(* Logix 5000 project; controller WWTP_SOLIDS_CLX vendor 1 type 14 code 54 rev 17.2; software revision 17.00; part 8 of 16 *)
(* tags used below, declared in another part *)
   PCmd_Tare : BOOL;   // Program Command to Tare (reset delivered qty to 0)
   PCmd_StartFlow : BOOL;   // Program Command to Start Delivery
   PCmd_StopFlow : BOOL;   // Program Command to Stop/Pause Delivery
   PCmd_CheckTol : BOOL;   // Program Command to Check Tolerances
   PCmd_OverTolInhibit : BOOL;   // Program Command to Inhibit Out of Tolerance High Alarm
   PCmd_OverTolUninhibit : BOOL;   // Program Command to Uninhibit Out of Tolerance High Alarm
   PCmd_UnderTolInhibit : BOOL;   // Program Command to Inhibit Out of Tolerance Low Alarm
   PCmd_UnderTolUninhibit : BOOL;   // Program Command to Uninhibit Out of Tolerance Low Alarm
   PCmd_TareFaultInhibit : BOOL;   // Program Command to Inhibit Tare Fault Alarm
   PCmd_TareFaultUninhibit : BOOL;   // Program Command to Uninhibit Tare Fault Alarm
   PCmd_EqpFaultInhibit : BOOL;   // Program Command to Inhibit Equipment Fault Alarm
   PCmd_EqpFaultUninhibit : BOOL;   // Program Command to Uninhibit Equipment Fault Alarm
   OCmd_Tare : BOOL;   // Operator Command to Tare (reset delivered qty to 0)
   OCmd_StartFlow : BOOL;   // Operator command to Start Deliver
   OCmd_StopFlow : BOOL;   // Operator Command to Stop/Pause Delivery
   OCmd_CheckTol : BOOL;   // Operator Command to Check Tolerances
   OCmd_Bump : BOOL;   // Operator Command to Bump Delivery for Under Tolerance
   Rdy_Tare : BOOL;   // 1=Ready for OCmd_Tare (enables button)
   Rdy_StartFlow : BOOL;   // 1=Ready for OCmd_StartFlow (enables button)
   Rdy_StopFlow : BOOL;   // 1=Ready for OCmd_StopFlow (enables button)
   Rdy_CheckTol : BOOL;   // 1-Ready for OCmd_CheckTol (enables button)
   Rdy_Bump : BOOL;   // 1=Ready for OCmd_Bump (enables button)
   Wrk_ValidONS1 : BOOL;   // Weight PV goes from Infinite or Not a Number to VALID
   Wrk_ValidONS2 : BOOL;   // Rate goes from Infinite or Not a Number to VALID
(* P_DoseWS, continued *)

ROUTINE Prescan   (* ladder *)
// Clear Ownership, clear "lurking" Commands, all Readies
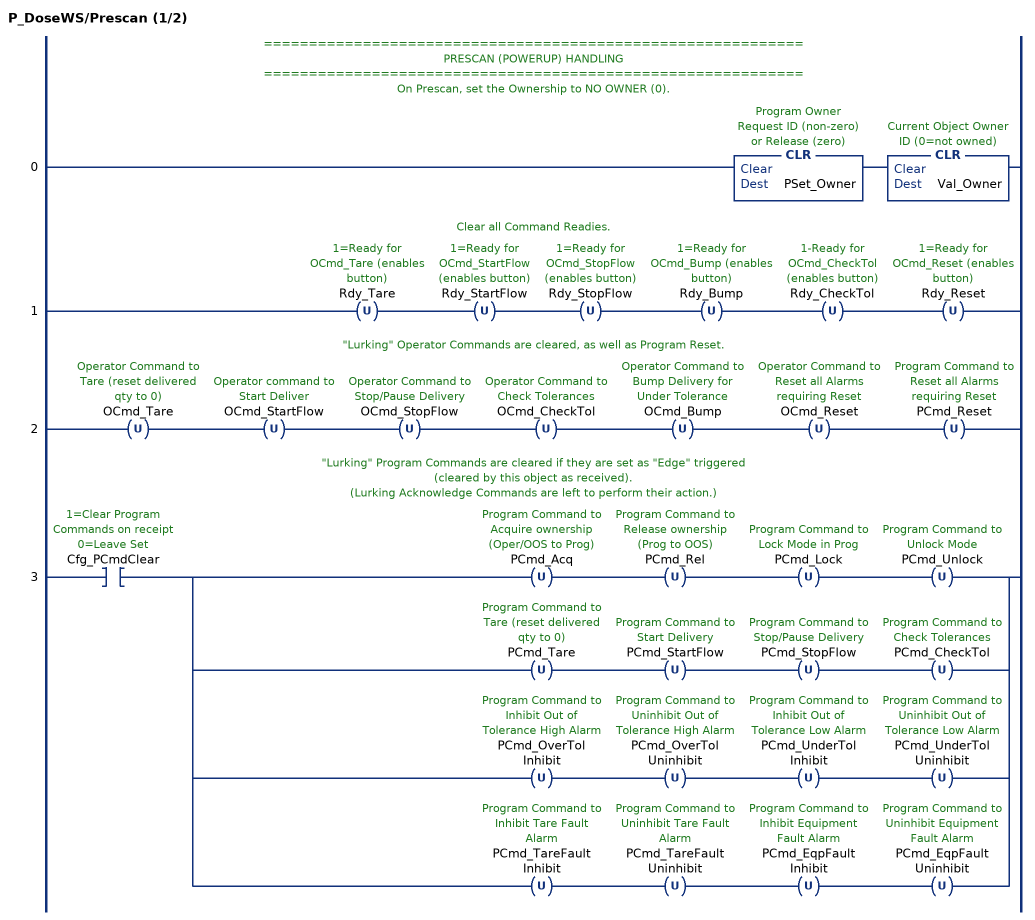
   // ============================================================
   // PRESCAN (POWERUP) HANDLING
   // ============================================================
   // On Prescan, set the Ownership to NO OWNER (0).
   0: CLR(PSet_Owner)CLR(Val_Owner);
   // Clear all Command Readies.
   1: OTU(Rdy_Tare)OTU(Rdy_StartFlow)OTU(Rdy_StopFlow)OTU(Rdy_Bump)OTU(Rdy_CheckTol)OTU(Rdy_Reset);
   // "Lurking" Operator Commands are cleared, as well as Program Reset.
   2: OTU(OCmd_Tare)OTU(OCmd_StartFlow)OTU(OCmd_StopFlow)OTU(OCmd_CheckTol)OTU(OCmd_Bump)OTU(OCmd_Reset)OTU(PCmd_Reset);
   // "Lurking" Program Commands are cleared if they are set as "Edge" triggered
   // (cleared by this object as received).
   // (Lurking Acknowledge Commands are left to perform their action.)
   3: XIC(Cfg_PCmdClear)[OTU(PCmd_Acq) OTU(PCmd_Rel) OTU(PCmd_Lock) OTU(PCmd_Unlock) ,OTU(PCmd_Tare) OTU(PCmd_StartFlow) OTU(PCmd_StopFlow) OTU(PCmd_CheckTol) ,OTU(PCmd_OverTolInhibit) OTU(PCmd_OverTolUninhibit) OTU(PCmd_UnderTolInhibit) OTU(PCmd_UnderTolUninhibit) ,OTU(PCmd_TareFaultInhibit) OTU(PCmd_TareFaultUninhibit) OTU(PCmd_EqpFaultInhibit) OTU(PCmd_EqpFaultUninhibit) ];
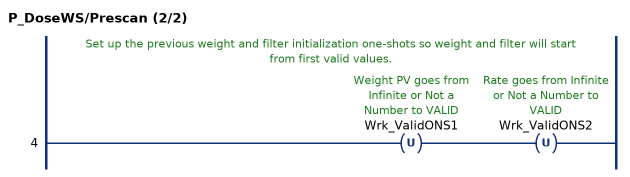
   // Set up the previous weight and filter initialization one-shots so weight and filter will start from first valid values.
   4: OTU(Wrk_ValidONS1)OTU(Wrk_ValidONS2);
END_ROUTINE
END_ADD_ON_INSTRUCTION

ADD_ON_INSTRUCTION P_Intlk   (* revision 0.10, ExecuteEnableInFalse *)
// Interlocks
// Revision note:
// Aligned name, description and local STRING values, sizes, across instructions.
// Help:
// This Instruction monitors up to 16 Interlock conditions.  It provides these features:
// *  Interlocks may be configured as Latched.
//     Latched Interlocks require a Reset Command to clear.
// *  Interlocks may be configured as Bypassable; Non-Bypassable
//     Interlocks are reported separately so the destination object can
//     decide whether to bypass (ignore) bypassable interlocks, such
//     as in Maintenance Mode.
// *  First-Out reporting indicates the first condition that caused the
//     running equipment to be tripped.  A separate First-Out is provided
//     for Non-Bypassable Interlocks.
VAR_INPUT
   Inp_Intlk00 : BOOL; {visible}   // Interlock Cond. 00 (1=Stop, 0=OK)
   Inp_Intlk01 : BOOL; {visible}   // Interlock Cond. 01 (1=Stop, 0=OK)
   Inp_Intlk02 : BOOL; {visible}   // Interlock Cond. 02 (1=Stop, 0=OK)
   Inp_Intlk03 : BOOL; {visible}   // Interlock Cond. 03 (1=Stop, 0=OK)
   Inp_Intlk04 : BOOL; {visible}   // Interlock Cond. 04 (1=Stop, 0=OK)
   Inp_Intlk05 : BOOL; {visible}   // Interlock Cond. 05 (1=Stop, 0=OK)
   Inp_Intlk06 : BOOL; {visible}   // Interlock Cond. 06 (1=Stop, 0=OK)
   Inp_Intlk07 : BOOL; {visible}   // Interlock Cond. 07 (1=Stop, 0=OK)
   Inp_Intlk08 : BOOL;   // Interlock Cond. 08 (1=Stop, 0=OK)
   Inp_Intlk09 : BOOL;   // Interlock Cond. 09 (1=Stop, 0=OK)
   Inp_Intlk10 : BOOL;   // Interlock Cond. 10 (1=Stop, 0=OK)
   Inp_Intlk11 : BOOL;   // Interlock Cond. 11 (1=Stop, 0=OK)
   Inp_Intlk12 : BOOL;   // Interlock Cond. 12 (1=Stop, 0=OK)
   Inp_Intlk13 : BOOL;   // Interlock Cond. 13 (1=Stop, 0=OK)
   Inp_Intlk14 : BOOL;   // Interlock Cond. 14 (1=Stop, 0=OK)
   Inp_Intlk15 : BOOL;   // Interlock Cond. 15 (1=Stop, 0=OK)
   Inp_Reset : BOOL; {visible}   // 1=Reset Latched Interlocks and First-Out
   Cfg_Latched : INT;   // Set bits indicate which conditions are latched (sealed in)
   Cfg_Bypassable : INT;   // Set bits indicate which conditions can be bypassed
   Cfg_PCmdClear : BOOL := 1;   // 1=Clear Program Commands on receipt 0=Leave Set
   PCmd_Reset : BOOL;   // Program Command to Reset Latched Interlocks
   OCmd_Reset : BOOL;   // Operator Command to Reset Latched Interlocks
END_VAR
VAR_OUTPUT
   Sts_IntlkOK : BOOL := 1; {visible}   // Overall Interlock Status (1=OK to run, 0=Stop)
   Sts_NBIntlkOK : BOOL := 1; {visible}   // Non-Bypassable Interlock Status (1=All NB Interlocks OK to run)
   Sts_Intlk : INT; {visible}   // Individual Interlock Status (1=Stop, 0=OK)
   Sts_FirstOut : INT; {visible}   // Interlock First Out Status (bit 1 is First Not-OK condition)
   Sts_NBFirstOut : INT; {visible}   // Non-bypassable Interlock First-Out Status (bit=1 is First NB Not-OK condition)
   Rdy_Reset : BOOL;   // 1=Ready to receive OCmd_Reset (reset required)
END_VAR
VAR
   Cfg_CondTxt : STRING_20[16] := ([0] := 'Interlock 0');   // Short HMI description of Interlock Conditions
   Wrk_Inp : INT;   // Collection copy of Inp_IntlkXXs
   Wrk_NB : INT;   // Working register for Non-Bypassable Interlock ogic
   Wrk_Intlk : INT;   // Working register for Interlock logic
   Wrk_FirstOut : INT;   // Working register for First Out logic
   Wrk_Sts : INT;   // Working register for generating Interlock status
   Wrk_NBFirstOut : INT;   // Working register for Non-Bypassable First Out logic
   Wrk_PrevSts : INT;   // Interlock Status previous scan
   Wrk_PrevNB : INT;   // Non-Bypassable Status previous scan
END_VAR

ROUTINE EnableInFalse   (* ladder *)
// Set summary "OK" Status bits to FALSE (0)
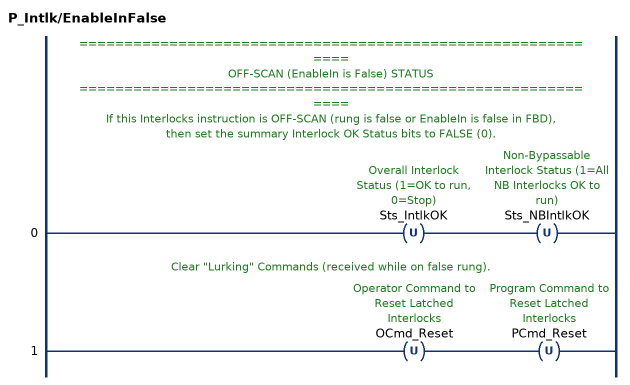
   // ============================================================
   // OFF-SCAN (EnableIn is False) STATUS
   // ============================================================
   // If this Interlocks instruction is OFF-SCAN (rung is false or EnableIn is false in FBD),
   // then set the summary Interlock OK Status bits to FALSE (0).
   0: OTU(Sts_IntlkOK)OTU(Sts_NBIntlkOK);
   // Clear "Lurking" Commands (received while on false rung).
   1: OTU(OCmd_Reset)OTU(PCmd_Reset);
END_ROUTINE

ROUTINE Logic   (* ladder *)
// Check Interlock Conditions
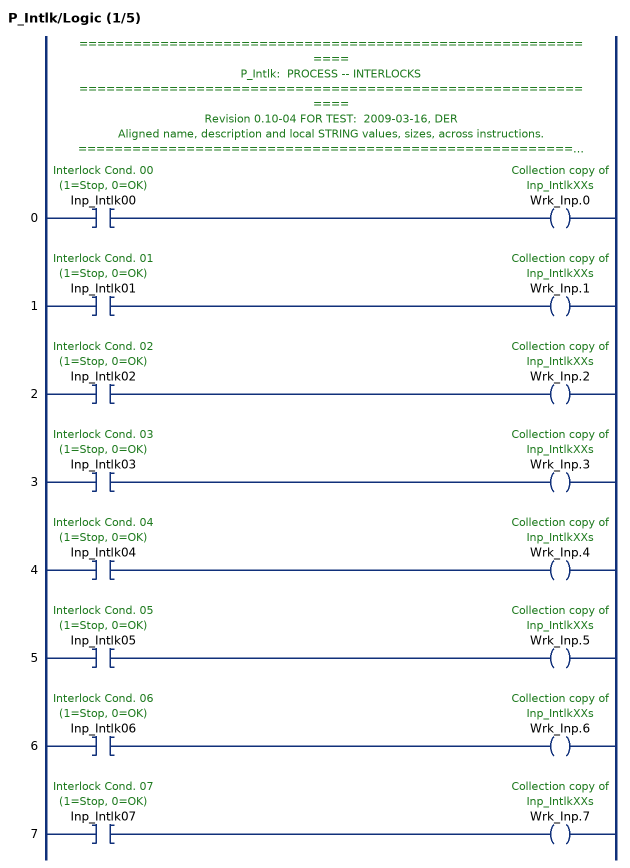
   // ============================================================
   // P_Intlk:  PROCESS -- INTERLOCKS
   // ============================================================
   // Revision 0.10-04 FOR TEST:  2009-03-16, DER
   // Aligned name, description and local STRING values, sizes, across instructions.
   // ============================================================
   // This Instruction monitors up to 16 Interlock conditions.  It provides these features:
   // *  Interlocks may be configured as Latched.  Latched Interlocks
   // require a Reset Command to clear.
   // *  Interlocks may be configured as Bypassable.  Bypassable Interlocks are reported
   // separately; the destination object can use this information to bypass these
   // Interlocks in Maintenance Mode or upon command.
   // *  First-Out reporting indicates the first condition that caused the running equipment
   // to be tripped.  Separate First-Out for Non-Bypassable Interlocks.
   // ============================================================
   // POWERUP / INVALID STATE HANDLING
   // ============================================================
   // Interlock, bypass and lock states are maintained through a power cycle or
   // run/prog/run cycle. No special powerup code is required for this object.
   // ============================================================
   // INPUT GATHERING
   // ============================================================
   // This object uses word-wise logic.  The first 16 rungs collect the individual
   // Interlock Inputs together into a 16-bit integer word for word-wise processing.
   0: XIC(Inp_Intlk00)OTE(Wrk_Inp.0);
   1: XIC(Inp_Intlk01)OTE(Wrk_Inp.1);
   2: XIC(Inp_Intlk02)OTE(Wrk_Inp.2);
   3: XIC(Inp_Intlk03)OTE(Wrk_Inp.3);
   4: XIC(Inp_Intlk04)OTE(Wrk_Inp.4);
   5: XIC(Inp_Intlk05)OTE(Wrk_Inp.5);
   6: XIC(Inp_Intlk06)OTE(Wrk_Inp.6);
   7: XIC(Inp_Intlk07)OTE(Wrk_Inp.7);
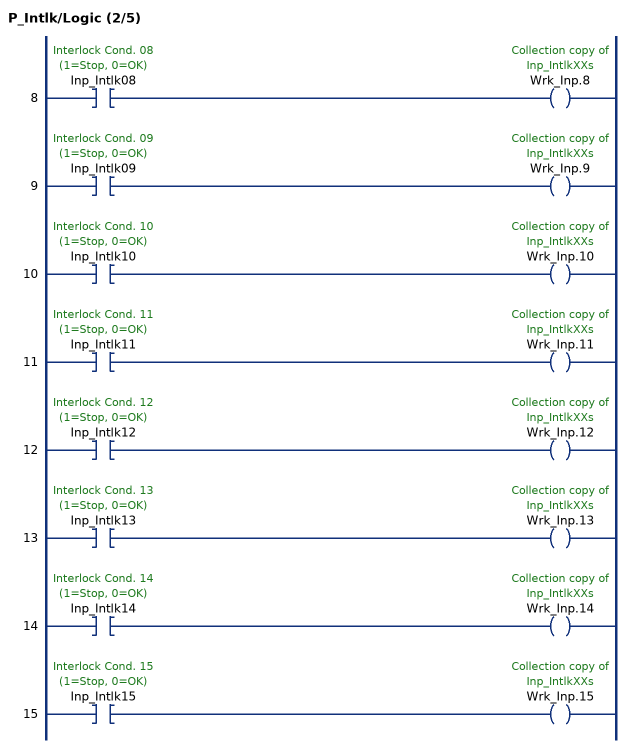
   8: XIC(Inp_Intlk08)OTE(Wrk_Inp.8);
   9: XIC(Inp_Intlk09)OTE(Wrk_Inp.9);
   10: XIC(Inp_Intlk10)OTE(Wrk_Inp.10);
   11: XIC(Inp_Intlk11)OTE(Wrk_Inp.11);
   12: XIC(Inp_Intlk12)OTE(Wrk_Inp.12);
   13: XIC(Inp_Intlk13)OTE(Wrk_Inp.13);
   14: XIC(Inp_Intlk14)OTE(Wrk_Inp.14);
   15: XIC(Inp_Intlk15)OTE(Wrk_Inp.15);
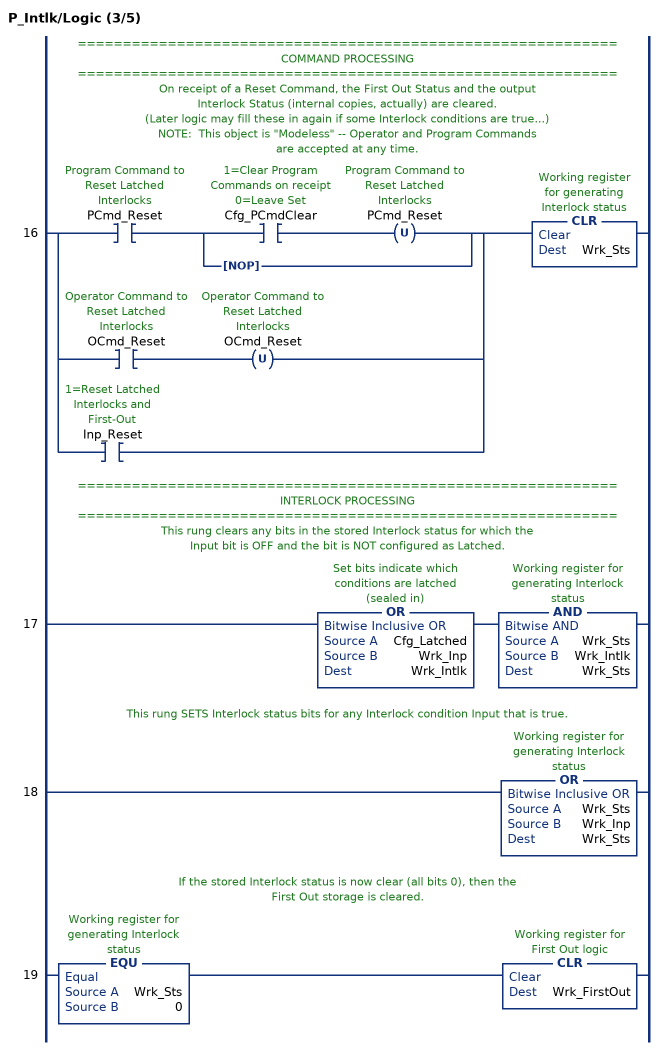
   // ============================================================
   // COMMAND PROCESSING
   // ============================================================
   // On receipt of a Reset Command, the First Out Status and the output
   // Interlock Status (internal copies, actually) are cleared.
   // (Later logic may fill these in again if some Interlock conditions are true...)
   // NOTE:  This object is "Modeless" -- Operator and Program Commands
   // are accepted at any time.
   16: [XIC(PCmd_Reset) [XIC(Cfg_PCmdClear) OTU(PCmd_Reset) ,NOP() ] ,XIC(OCmd_Reset) OTU(OCmd_Reset) ,XIC(Inp_Reset) ]CLR(Wrk_Sts);
   // ============================================================
   // INTERLOCK PROCESSING
   // ============================================================
   // This rung clears any bits in the stored Interlock status for which the
   // Input bit is OFF and the bit is NOT configured as Latched.
   17: OR(Cfg_Latched,Wrk_Inp,Wrk_Intlk)AND(Wrk_Sts,Wrk_Intlk,Wrk_Sts);
   // This rung SETS Interlock status bits for any Interlock condition Input that is true.
   18: OR(Wrk_Sts,Wrk_Inp,Wrk_Sts);
   // If the stored Interlock status is now clear (all bits 0), then the
   // First Out storage is cleared.
   19: EQU(Wrk_Sts,0)CLR(Wrk_FirstOut);
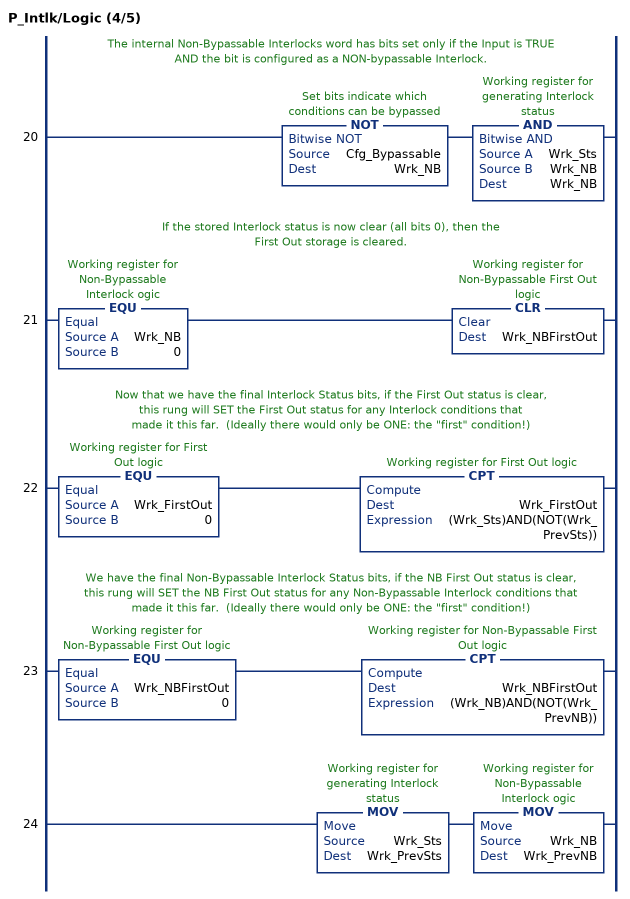
   // The internal Non-Bypassable Interlocks word has bits set only if the Input is TRUE
   // AND the bit is configured as a NON-bypassable Interlock.
   20: NOT(Cfg_Bypassable,Wrk_NB)AND(Wrk_Sts,Wrk_NB,Wrk_NB);
   // If the stored Interlock status is now clear (all bits 0), then the
   // First Out storage is cleared.
   21: EQU(Wrk_NB,0)CLR(Wrk_NBFirstOut);
   // Now that we have the final Interlock Status bits, if the First Out status is clear,
   // this rung will SET the First Out status for any Interlock conditions that
   // made it this far.  (Ideally there would only be ONE: the "first" condition!)
   22: EQU(Wrk_FirstOut,0)CPT(Wrk_FirstOut,(Wrk_Sts)AND(NOT(Wrk_PrevSts)));
   // We have the final Non-Bypassable Interlock Status bits, if the NB First Out status is clear,
   // this rung will SET the NB First Out status for any Non-Bypassable Interlock conditions that
   // made it this far.  (Ideally there would only be ONE: the "first" condition!)
   23: EQU(Wrk_NBFirstOut,0)CPT(Wrk_NBFirstOut,(Wrk_NB)AND(NOT(Wrk_PrevNB)));
   24: MOV(Wrk_Sts,Wrk_PrevSts)MOV(Wrk_NB,Wrk_PrevNB);
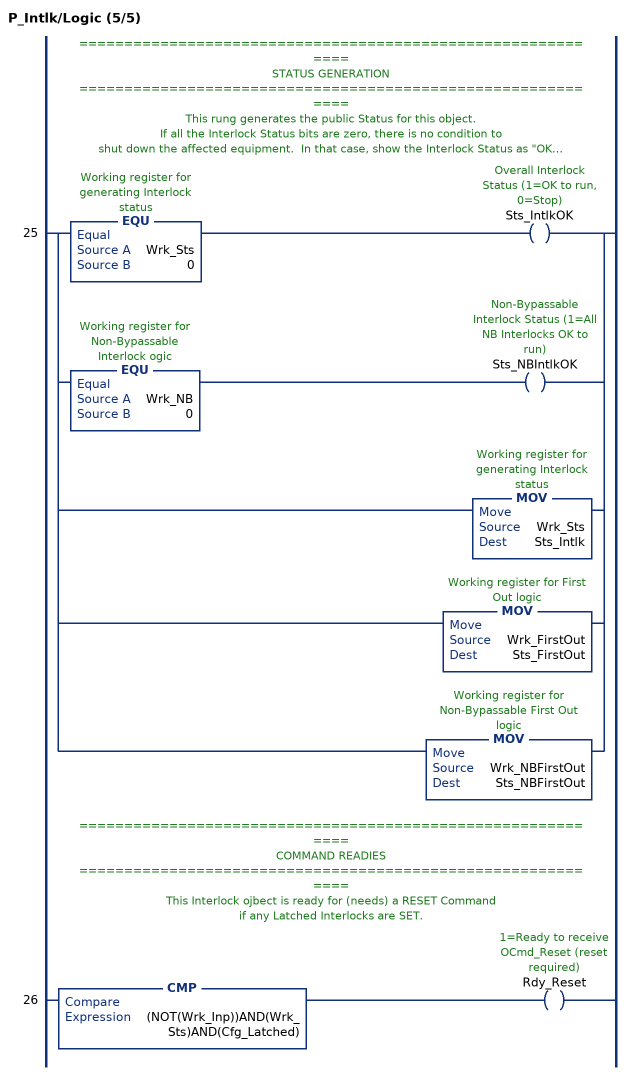
   // ============================================================
   // STATUS GENERATION
   // ============================================================
   // This rung generates the public Status for this object.
   // If all the Interlock Status bits are zero, there is no condition to
   // shut down the affected equipment.  In that case, show the Interlock Status as "OK"
   // Similar logic applies for the Non-Bypassable Interlocks OK Status.
   // Also show the individual Interlock Status bits and the First Out Status bits.
   // NOTE:  Working registers are used to prevent outside writes to the Sts_xxx
   // parameters from affecting the state of this object!
   25: [[EQU(Wrk_Sts,0) OTE(Sts_IntlkOK) ,EQU(Wrk_NB,0) OTE(Sts_NBIntlkOK) ] ,MOV(Wrk_Sts,Sts_Intlk) ,MOV(Wrk_FirstOut,Sts_FirstOut) ,MOV(Wrk_NBFirstOut,Sts_NBFirstOut) ];
   // ============================================================
   // COMMAND READIES
   // ============================================================
   // This Interlock ojbect is ready for (needs) a RESET Command
   // if any Latched Interlocks are SET.
   26: CMP((NOT(Wrk_Inp))AND(Wrk_Sts)AND(Cfg_Latched))OTE(Rdy_Reset);
END_ROUTINE

ROUTINE Prescan   (* ladder *)
// Clear "lurking" Commands
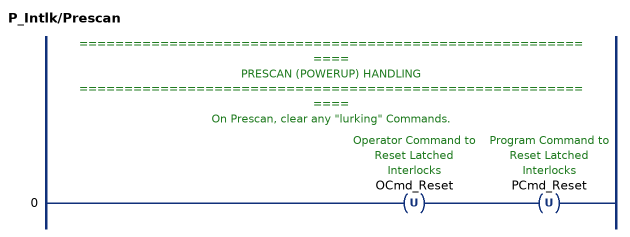
   // ============================================================
   // PRESCAN (POWERUP) HANDLING
   // ============================================================
   // On Prescan, clear any "lurking" Commands.
   0: OTU(OCmd_Reset)OTU(PCmd_Reset);
END_ROUTINE
END_ADD_ON_INSTRUCTION

ADD_ON_INSTRUCTION P_Mode   (* revision 0.20, ExecutePrescan, ExecuteEnableInFalse *)
// Mode
// Revision note:
// Aligned name, description and local STRING values, sizes, across instructions.
// Help:
// This instruction provides selection of Mode for a Device-level
//  object (motor, valve, drive, loop, etc.).  Possible Modes are:
//    Hand (typically tracks hardwired logic)
//    Maintenance (not available for operation)
//    Override (typically process or soft safety interlock logic)
//    Operator (settings and commands from HMI)
//    Program (settings and commands from other objects)
// Hand and Override are selected via Input parameters (pins).
// Program and Maintenance are acquired and released via Commands.
// Program or Operator owner can Lock ownership; when locked, Hand and
// Maintenance override the Lock.  Override can be configured as to
// whether or not it supersedes Locked Program or Operator ownership.
// Program Commands can be configured as one-shot (OTL) inputs (default),
// or Level-based inputs.  One-shot Program Commands are cleared by the
// Mode object; When Level-based, the Program Acquire (PCmd_Acq)
// Command is left set; when the Program clears this Command, Program Mode is
// released; and when the Program Lock (PCmd_Lock) command is cleared,
// Program Mode is unlocked.
// Program and Operator commands work "behind the scenes" while in Hand,
// Ovrd or Maint; so the Program can release the object while in Hand, and
// upon exiting Hand, the Mode will revert to Operator, for example.  Extra Status
// bits indicate the results of these "behind the scenes" activities.
VAR_INPUT
   Inp_Hand : BOOL; {visible}   // 1=Select Hand (typ. hardwired) Mode
   Inp_Ovrd : BOOL; {visible}   // 1=Select Override (typ. Process/Safety Interlock) Mode
   Cfg_PCmdClear : BOOL := 1;   // 1=Clear Program Command on receipt; 0=Use Level-based (maintained) PCmds
   Cfg_OvrdOverLock : BOOL := 1;   // 1=Override supersedes Prog/Oper Lock, 0=don't override Lock
   PCmd_Acq : BOOL;   // Program Command to Acquire Ownership (Oper to Prog)
   PCmd_Rel : BOOL;   // Program Command to Release Ownership (Prog to Oper)
   PCmd_Lock : BOOL;   // Program Command to Lock Mode in Prog
   PCmd_Unlock : BOOL;   // Program Command to Unlock Mode
   MCmd_Acq : BOOL;   // Maintenance Command to Acquire Ownership (Oper/Prog/Ovrd to Maint)
   MCmd_Rel : BOOL;   // Maintenance Command to Release Ownership (Maint to Oper/Prog/Ovrd)
   OCmd_AcqLock : BOOL;   // Operator Command to Acquire and Lock Mode in Oper
   OCmd_Unlock : BOOL;   // Operator Command to Unlock Operator Mode
END_VAR
VAR_OUTPUT
   Sts_Hand : BOOL; {visible}   // 1=Mode is Hand (supersedes Maint, Ovrd, Prog, Oper)
   Sts_Maint : BOOL; {visible}   // 1=Mode is Maintenance (supersedes Ovrd, Prog, Oper)
   Sts_Ovrd : BOOL; {visible}   // 1=Mode is Override (supersedes Prog, Oper)
   Sts_Prog : BOOL; {visible}   // 1=Mode is Program
   Sts_Oper : BOOL := 1; {visible}   // 1=Mode is Operator
   Sts_ProgOperLock : BOOL; {visible}   // 1=Program or Operator has requested Mode Lock
   Sts_ProgOperSel : BOOL;   // Prog/Oper selection 1=Program, 0=Operator
   Rdy_Acq : BOOL;   // 1=Ready for MCmd_Acq
   Rdy_Rel : BOOL;   // 1=Ready for MCmd_Rel
   Rdy_AcqLock : BOOL;   // 1=Ready for OCmd_AcqLock
   Rdy_Unlock : BOOL;   // 1=Ready for OCmd_Unlock
END_VAR
VAR
   Wrk_Locked : BOOL;   // 1=Program/Operator Mode selection is Locked
   Wrk_Prog : BOOL;   // Internal Program (1) / Operator (0) Mode selection
   Wrk_Maint : BOOL;   // Internal Maintenance Mode
END_VAR

ROUTINE EnableInFalse   (* ladder *)
// Processes received Commands, but shows NO owner
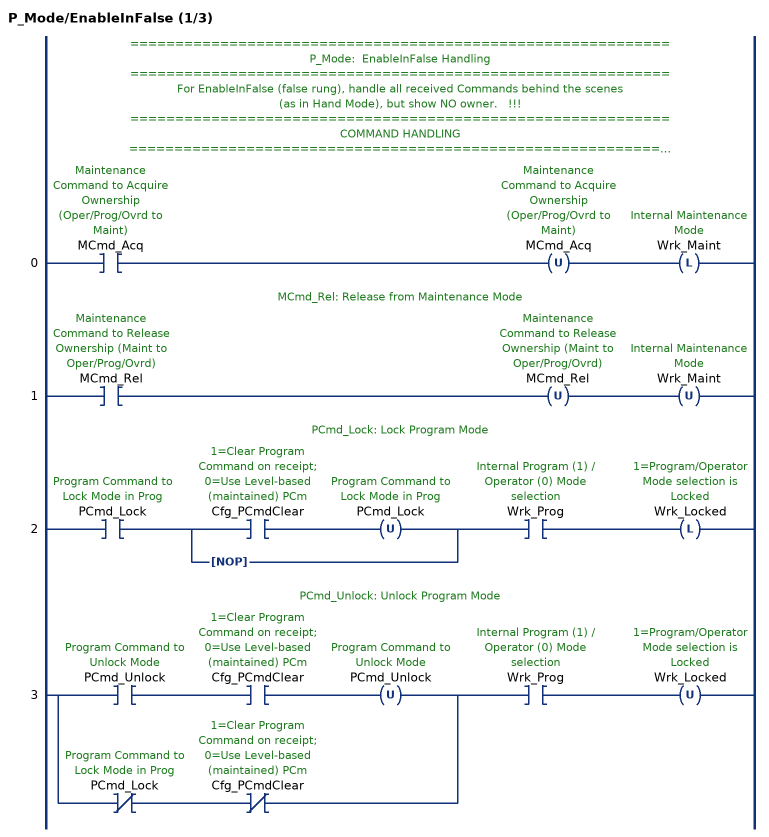
   // ============================================================
   // P_Mode:  EnableInFalse Handling
   // ============================================================
   // For EnableInFalse (false rung), handle all received Commands behind the scenes
   // (as in Hand Mode), but show NO owner.   !!!
   // ============================================================
   // COMMAND HANDLING
   // ============================================================
   // NOTE:  These rungs MUST be in the order given to meet the following
   // multiple-actions-at-the-same-time scenarios:
   // * Maintenance Release beats Maintenance Acquire
   // * Program Release beats Program Acquire
   // * Program Unlock beats Program Lock
   // * Operator Unlock beats Operator Acquire and Lock (results in Oper Unlocked)
   // * Operator Acquire/Lock must come after Program Unlock
   // * Program Acquire must come after Operator Unlock
   // MCmd_Acq: Acquire for Maintenance Mode
   0: XIC(MCmd_Acq)OTU(MCmd_Acq)OTL(Wrk_Maint);
   // MCmd_Rel: Release from Maintenance Mode
   1: XIC(MCmd_Rel)OTU(MCmd_Rel)OTU(Wrk_Maint);
   // PCmd_Lock: Lock Program Mode
   2: XIC(PCmd_Lock)[XIC(Cfg_PCmdClear) OTU(PCmd_Lock) ,NOP() ]XIC(Wrk_Prog)OTL(Wrk_Locked);
   // PCmd_Unlock: Unlock Program Mode
   3: [XIC(PCmd_Unlock) XIC(Cfg_PCmdClear) OTU(PCmd_Unlock) ,XIO(PCmd_Lock) XIO(Cfg_PCmdClear) ]XIC(Wrk_Prog)OTU(Wrk_Locked);
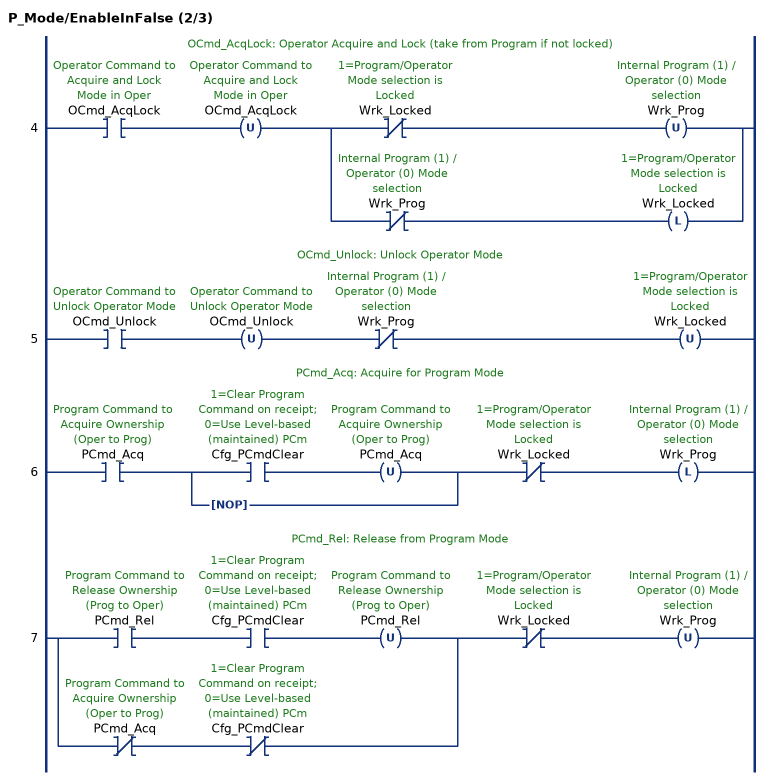
   // OCmd_AcqLock: Operator Acquire and Lock (take from Program if not locked)
   4: XIC(OCmd_AcqLock)OTU(OCmd_AcqLock)[XIO(Wrk_Locked) OTU(Wrk_Prog) ,XIO(Wrk_Prog) OTL(Wrk_Locked) ];
   // OCmd_Unlock: Unlock Operator Mode
   5: XIC(OCmd_Unlock)OTU(OCmd_Unlock)XIO(Wrk_Prog)OTU(Wrk_Locked);
   // PCmd_Acq: Acquire for Program Mode
   6: XIC(PCmd_Acq)[XIC(Cfg_PCmdClear) OTU(PCmd_Acq) ,NOP() ]XIO(Wrk_Locked)OTL(Wrk_Prog);
   // PCmd_Rel: Release from Program Mode
   7: [XIC(PCmd_Rel) XIC(Cfg_PCmdClear) OTU(PCmd_Rel) ,XIO(PCmd_Acq) XIO(Cfg_PCmdClear) ]XIO(Wrk_Locked)OTU(Wrk_Prog);
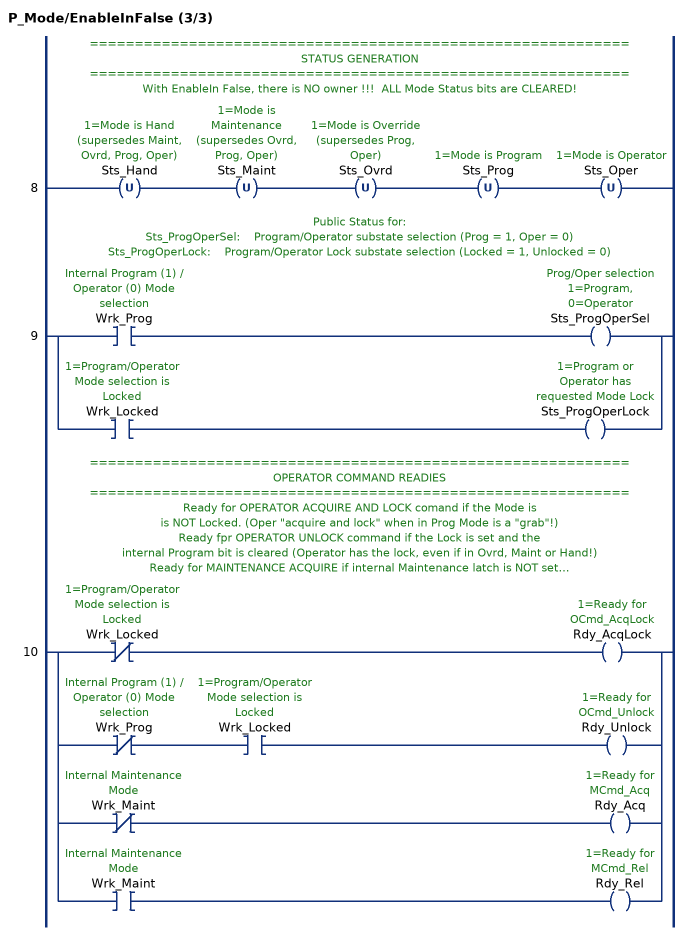
   // ============================================================
   // STATUS GENERATION
   // ============================================================
   // With EnableIn False, there is NO owner !!!  ALL Mode Status bits are CLEARED!
   8: OTU(Sts_Hand)OTU(Sts_Maint)OTU(Sts_Ovrd)OTU(Sts_Prog)OTU(Sts_Oper);
   // Public Status for:
   // Sts_ProgOperSel:    Program/Operator substate selection (Prog = 1, Oper = 0)
   // Sts_ProgOperLock:    Program/Operator Lock substate selection (Locked = 1, Unlocked = 0)
   9: [XIC(Wrk_Prog) OTE(Sts_ProgOperSel) ,XIC(Wrk_Locked) OTE(Sts_ProgOperLock) ];
   // ============================================================
   // OPERATOR COMMAND READIES
   // ============================================================
   // Ready for OPERATOR ACQUIRE AND LOCK comand if the Mode is
   //  is NOT Locked. (Oper "acquire and lock" when in Prog Mode is a "grab"!)
   // Ready fpr OPERATOR UNLOCK command if the Lock is set and the
   // internal Program bit is cleared (Operator has the lock, even if in Ovrd, Maint or Hand!)
   // Ready for MAINTENANCE ACQUIRE if internal Maintenance latch is NOT set.
   // Ready for MAINTENANCE RELEASE if internal Maintenance latch IS set.
   10: [XIO(Wrk_Locked) OTE(Rdy_AcqLock) ,XIO(Wrk_Prog) XIC(Wrk_Locked) OTE(Rdy_Unlock) ,XIO(Wrk_Maint) OTE(Rdy_Acq) ,XIC(Wrk_Maint) OTE(Rdy_Rel) ];
END_ROUTINE

ROUTINE Logic   (* ladder *)
// Selects Modes (Hand, Maint, Ovrd, Oper, Prog) based on Inputs and Commands
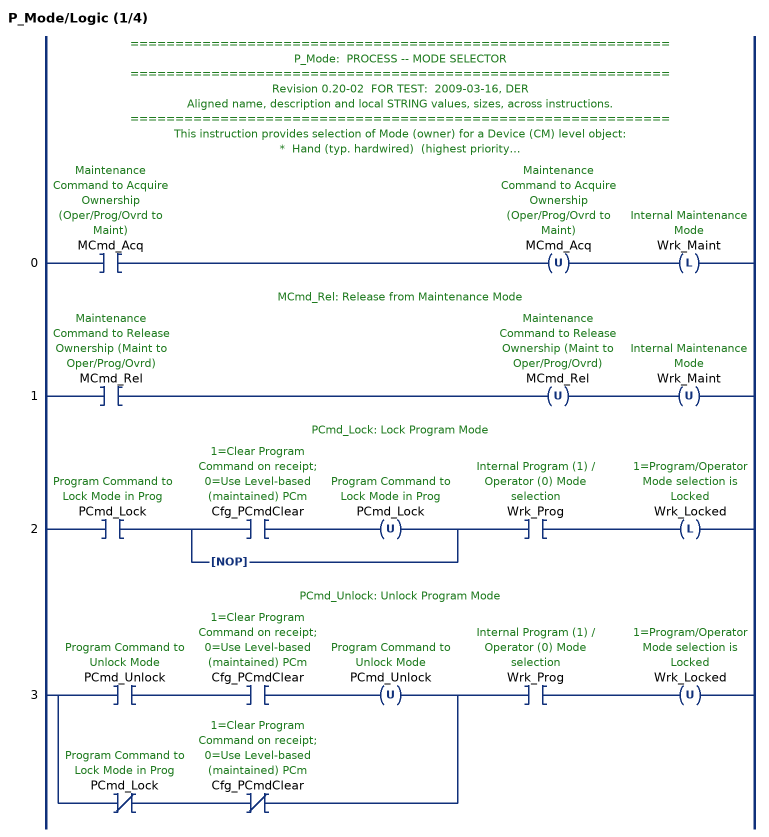
   // ============================================================
   // P_Mode:  PROCESS -- MODE SELECTOR
   // ============================================================
   // Revision 0.20-02  FOR TEST:  2009-03-16, DER
   // Aligned name, description and local STRING values, sizes, across instructions.
   // ============================================================
   // This instruction provides selection of Mode (owner) for a Device (CM) level object:
   // *  Hand (typ. hardwired)  (highest priority)
   // *  Maint (taken out of service for maintenance)
   // *  Ovrd (typ. process or soft safety interlock)
   // *  Prog  (automated control)
   // *  Oper (manual control)  (lowest priority owner)
   // ============================================================
   // COMMAND HANDLING
   // ============================================================
   // NOTE:  These rungs MUST be in the order given to meet the following
   // multiple-actions-at-the-same-time scenarios:
   // * Maintenance Release beats Maintenance Acquire
   // * Program Release beats Program Acquire
   // * Program Unlock beats Program Lock
   // * Operator Unlock beats Operator Acquire and Lock (results in Oper Unlocked)
   // * Operator Acquire/Lock must come after Program Unlock
   // * Program Acquire must come after Operator Unlock
   // MCmd_Acq: Acquire for Maintenance Mode
   0: XIC(MCmd_Acq)OTU(MCmd_Acq)OTL(Wrk_Maint);
   // MCmd_Rel: Release from Maintenance Mode
   1: XIC(MCmd_Rel)OTU(MCmd_Rel)OTU(Wrk_Maint);
   // PCmd_Lock: Lock Program Mode
   2: XIC(PCmd_Lock)[XIC(Cfg_PCmdClear) OTU(PCmd_Lock) ,NOP() ]XIC(Wrk_Prog)OTL(Wrk_Locked);
   // PCmd_Unlock: Unlock Program Mode
   3: [XIC(PCmd_Unlock) XIC(Cfg_PCmdClear) OTU(PCmd_Unlock) ,XIO(PCmd_Lock) XIO(Cfg_PCmdClear) ]XIC(Wrk_Prog)OTU(Wrk_Locked);
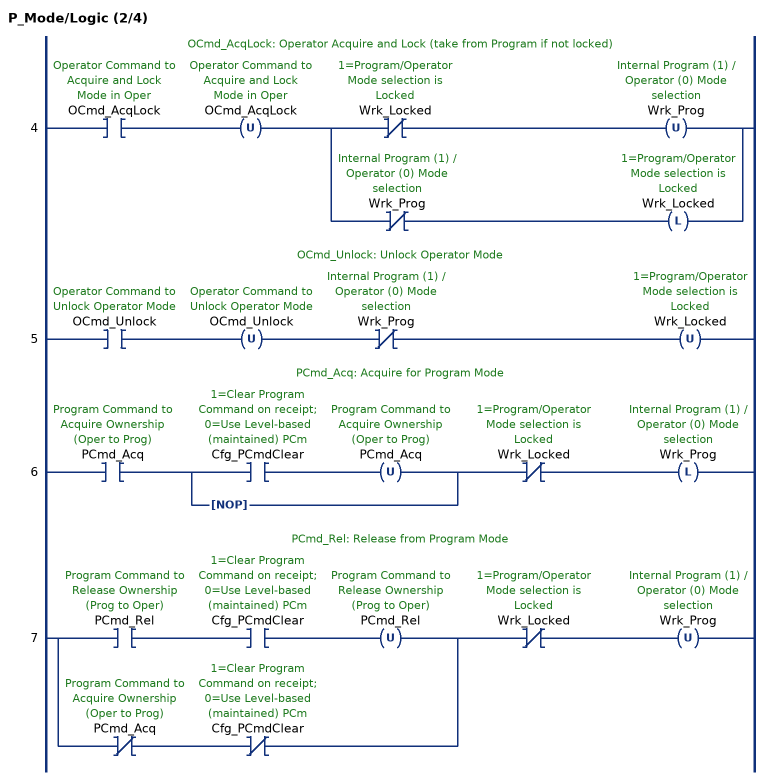
   // OCmd_AcqLock: Operator Acquire and Lock (take from Program if not locked)
   4: XIC(OCmd_AcqLock)OTU(OCmd_AcqLock)[XIO(Wrk_Locked) OTU(Wrk_Prog) ,XIO(Wrk_Prog) OTL(Wrk_Locked) ];
   // OCmd_Unlock: Unlock Operator Mode
   5: XIC(OCmd_Unlock)OTU(OCmd_Unlock)XIO(Wrk_Prog)OTU(Wrk_Locked);
   // PCmd_Acq: Acquire for Program Mode
   6: XIC(PCmd_Acq)[XIC(Cfg_PCmdClear) OTU(PCmd_Acq) ,NOP() ]XIO(Wrk_Locked)OTL(Wrk_Prog);
   // PCmd_Rel: Release from Program Mode
   7: [XIC(PCmd_Rel) XIC(Cfg_PCmdClear) OTU(PCmd_Rel) ,XIO(PCmd_Acq) XIO(Cfg_PCmdClear) ]XIO(Wrk_Locked)OTU(Wrk_Prog);
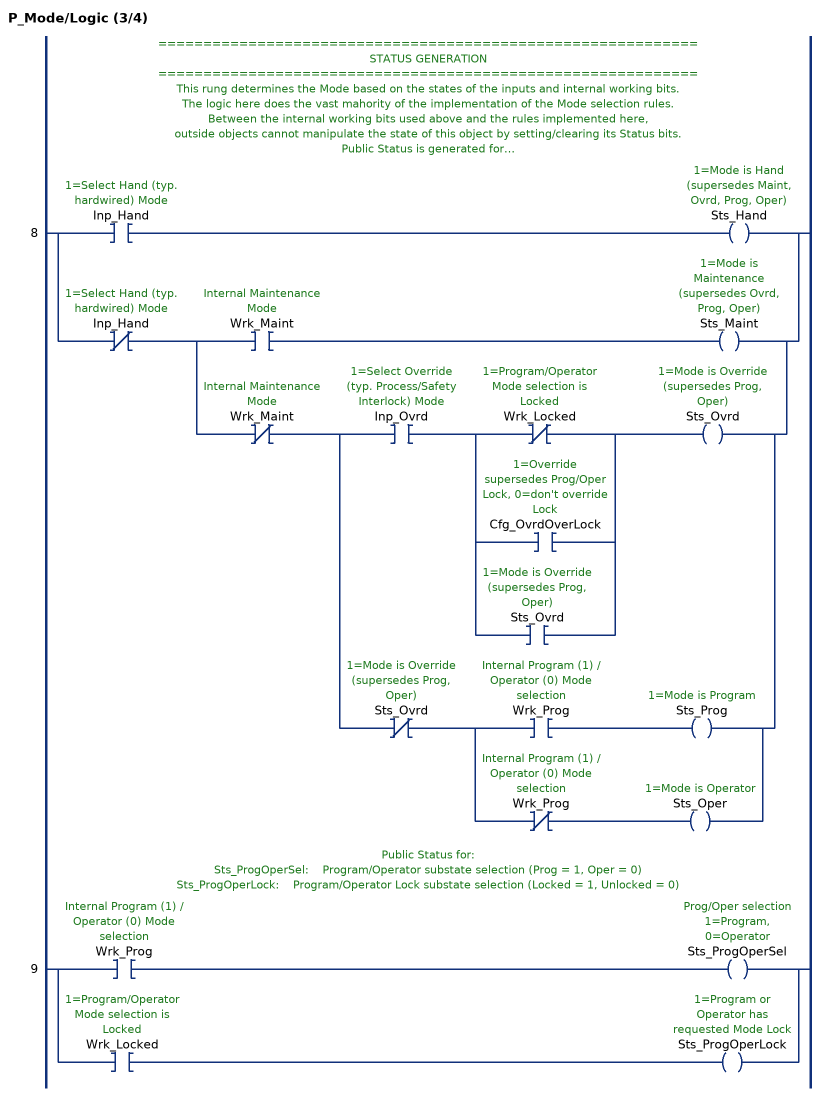
   // ============================================================
   // STATUS GENERATION
   // ============================================================
   // This rung determines the Mode based on the states of the inputs and internal working bits.
   // The logic here does the vast mahority of the implementation of the Mode selection rules.
   // Between the internal working bits used above and the rules implemented here,
   // outside objects cannot manipulate the state of this object by setting/clearing its Status bits.
   // Public Status is generated for:
   // *  Hand Mode
   // *  Maintenance Mode
   // *  Override Mode
   // *  Program Mode
   // *  Operator Mode
   8: [XIC(Inp_Hand) OTE(Sts_Hand) ,XIO(Inp_Hand) [XIC(Wrk_Maint) OTE(Sts_Maint) ,XIO(Wrk_Maint) [XIC(Inp_Ovrd) [XIO(Wrk_Locked) ,XIC(Cfg_OvrdOverLock) ,XIC(Sts_Ovrd) ] OTE(Sts_Ovrd) ,XIO(Sts_Ovrd) [XIC(Wrk_Prog) OTE(Sts_Prog) ,XIO(Wrk_Prog) OTE(Sts_Oper) ] ] ] ];
   // Public Status for:
   // Sts_ProgOperSel:    Program/Operator substate selection (Prog = 1, Oper = 0)
   // Sts_ProgOperLock:    Program/Operator Lock substate selection (Locked = 1, Unlocked = 0)
   9: [XIC(Wrk_Prog) OTE(Sts_ProgOperSel) ,XIC(Wrk_Locked) OTE(Sts_ProgOperLock) ];
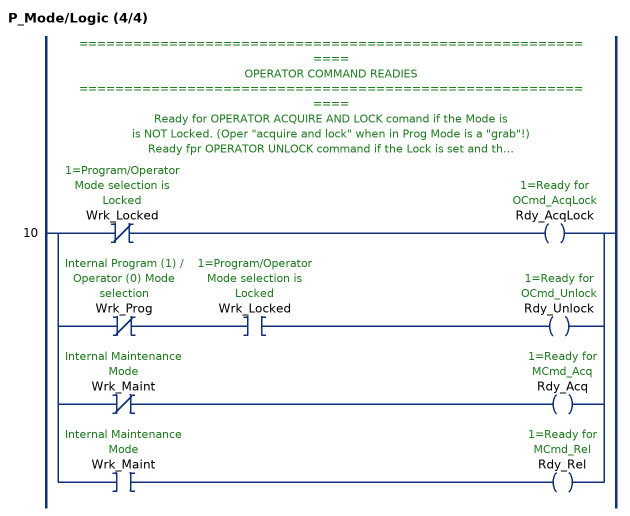
   // ============================================================
   // OPERATOR COMMAND READIES
   // ============================================================
   // Ready for OPERATOR ACQUIRE AND LOCK comand if the Mode is
   //  is NOT Locked. (Oper "acquire and lock" when in Prog Mode is a "grab"!)
   // Ready fpr OPERATOR UNLOCK command if the Lock is set and the
   // internal Program bit is cleared (Operator has the lock, even if in Ovrd, Maint or Hand!)
   // Ready for MAINTENANCE ACQUIRE if internal Maintenance latch is NOT set.
   // Ready for MAINTENANCE RELEASE if internal Maintenance latch IS set.
   10: [XIO(Wrk_Locked) OTE(Rdy_AcqLock) ,XIO(Wrk_Prog) XIC(Wrk_Locked) OTE(Rdy_Unlock) ,XIO(Wrk_Maint) OTE(Rdy_Acq) ,XIC(Wrk_Maint) OTE(Rdy_Rel) ];
END_ROUTINE

ROUTINE Prescan   (* ladder *)
// Clear "lurking" Commands
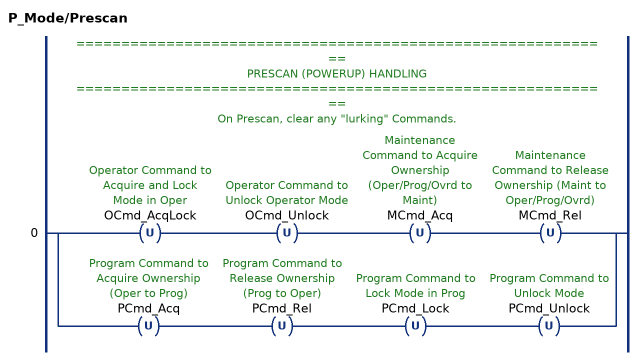
   // ============================================================
   // PRESCAN (POWERUP) HANDLING
   // ============================================================
   // On Prescan, clear any "lurking" Commands.
   0: [OTU(OCmd_AcqLock) OTU(OCmd_Unlock) OTU(MCmd_Acq) OTU(MCmd_Rel) ,OTU(PCmd_Acq) OTU(PCmd_Rel) OTU(PCmd_Lock) OTU(PCmd_Unlock) ];
END_ROUTINE
END_ADD_ON_INSTRUCTION

ADD_ON_INSTRUCTION P_Motor   (* revision 0.34, ExecutePrescan, ExecuteEnableInFalse *)
// Single Speed Motor
// Revision note:
// Aligned name, description and local STRING values, sizes, across instructions.
// Help:
// This Instruction controls and monitors a single-speed motor
// (FVNR, soft-start, etc.) and provides:
// *  Monitoring of run feedback, display of actual motor status
// *  Detection of Failure to Start, Failure to Stop
// *  Monitoring of Permissive conditions to allow starting
// *  Monitoring of Interlock conditions to stop / prevent starting
// *  Simulation, providing feedback of a working motor while disabling outputs
// *  Monitoring of I/O communication faults
// *  Alarms for Fail to Start, Fail to Stop, Interlock Trip, I/O Fault
// *  Operation in Hand, Maintenance, Override, Program and Operator Modes
// *  "Available" status for use by automation logic to know whether motor
//       can be controlled by other objects.
VAR_INPUT
   Inp_RunFdbk : BOOL; {visible}   // Input Signal: RUN feedback from motor
   Inp_PermOK : BOOL := 1; {visible}   // 1=Permissives OK, motor can start
   Inp_NBPermOK : BOOL := 1; {visible}   // 1=Non-Bypassable Permissives OK, motor can start
   Inp_IntlkOK : BOOL := 1; {visible}   // 1=Interlocks OK, motor can start/run
   Inp_NBIntlkOK : BOOL := 1; {visible}   // 1=Non-Bypassable Interlocks OK, motor can start/run
   Inp_IOFault : BOOL;   // Input Communication Status 0=OK, 1=fail
   Inp_Sim : BOOL;   // 1=Simulate working motor; 0=Start/Stop/ Monitor actual motor
   Inp_Hand : BOOL;   // 1=Select Hand (hardwired) Control Strategy
   Inp_Ovrd : BOOL;   // 1=Select Override control strategy
   Inp_OvrdState : BOOL;   // 1=Override to RUN, 0=Override to STOP
   Inp_Reset : BOOL;   // 1=Reset all fault conditions and latched Alarms
   Cfg_HasRunFdbk : BOOL;   // 1=Motor provides a run feedback signal
   Cfg_UseRunFdbk : BOOL;   // 1=Motor run feedback should be used for failure checking
   Cfg_HasPermObj : BOOL;   // 1=Tells HMI a P_Perm is connected to Inp_Perm
   Cfg_HasIntlkObj : BOOL;   // 1=Tells HMI a P_Intlk is connected to Inp_Intlk
   Cfg_HasResInhObj : BOOL;   // 1=Tells HMI a P_ResInh Restart Inhibit is connected
   Cfg_HasRunTimeObj : BOOL;   // 1=Tells HMI a P_RunTime is connected
   Cfg_PCmdClear : BOOL := 1;   // 1=Clear Program Commands on receipt 0=Leave Set
   Cfg_OvrdPermIntlk : BOOL;   // 1=Override ignores Bypassable Perm/ Intlk; 0=always use Perm/Intlk
   Cfg_HasFailToStartAlm : BOOL;   // 1=Fail to Start Alarm exists and will be checked
   Cfg_HasFailToStopAlm : BOOL;   // 1=Fail to Stop Alarm exists and will be checked
   Cfg_HasIntlkTripAlm : BOOL;   // 1=Interlock Trip Alarm exists and will be checked
   Cfg_HasIOFaultAlm : BOOL;   // 1=I/O Fault Alarm exists and will be checked
   Cfg_FailToStartResetReqd : BOOL;   // 1=Reset required to clear Fail to Start Alarm
   Cfg_FailToStopResetReqd : BOOL;   // 1=Reset required to clear Fail to Stop Alarm
   Cfg_IntlkTripResetReqd : BOOL;   // 1=Reset required to clear Interlock Trip Alarm
   Cfg_IOFaultResetReqd : BOOL;   // 1=Reset required to clear I/O Fault Alarm
   Cfg_FailToStartAckReqd : BOOL := 1;   // 1=Acknowledge required for Fail to Start Alarm
   Cfg_FailToStopAckReqd : BOOL := 1;   // 1=Acknowledge required for Fail to Stop Alarm
   Cfg_IntlkTripAckReqd : BOOL := 1;   // 1=Acknowledge required for Interlock Trip Alarm
   Cfg_IOFaultAckReqd : BOOL := 1;   // 1=Acknowledge required for I/O Fault Alarm
   Cfg_FailToStartSeverity : SINT := 4;   // Fail To Start Alarm Severity 1=info 2=warn 3=excep 4=fault
   Cfg_FailToStopSeverity : SINT := 4;   // Fail To Stop Alarm Severity 1=info 2=warn 3=excep 4=fault
   Cfg_IntlkTripSeverity : SINT := 2;   // Interlock Trip Alarm Severity 1=info 2=warn 3=excep 4=fault
   Cfg_IOFaultSeverity : SINT := 4;   // I/O Fault Alarm Severity 1=info 2=warn 3=excep 4=fault
   Cfg_SimFdbkT : DINT := 2;   // Delay to echo back of Running/Stopped status when in Simulation (sec)
   Cfg_FailToStartT : DINT := 10;   // Time after Start to get Run Feedback before Fault (sec)
   Cfg_FailToStopT : DINT := 10;   // Time after Stop to drop Run Feedback before Fault (sec)
   PSet_Owner : DINT;   // Program Owner Request ID (non-zero) or Release (zero)
   PCmd_Start : BOOL;   // Program Command to Start Motor
   PCmd_Stop : BOOL;   // Program Command to Stop Motor
   PCmd_Acq : BOOL;   // Program Command to Acquire ownership (Oper/OOS to Prog)
   PCmd_Rel : BOOL;   // Program Command to Release ownership (Prog to OOS)
   PCmd_Lock : BOOL;   // Program Command to Lock Mode in Prog
   PCmd_Unlock : BOOL;   // Program Command to Unlock Mode
   PCmd_Reset : BOOL;   // Program Command to Reset all Alarms requiring Reset
   PCmd_FailToStartAck : BOOL;   // Program Command to Acknowledge Fail to Start Alarm
   PCmd_FailToStartInhibit : BOOL;   // Program Command to Inhibit Fail to Start Alarm
   PCmd_FailToStartUninhibit : BOOL;   // Program Command to Uninhibit Fail to Start Alarm
   PCmd_FailToStopAck : BOOL;   // Program Command to Acknowledge Fail to Stop Alarm
   PCmd_FailToStopInhibit : BOOL;   // Program Command to Inhibit Fail to Stop Alarm
   PCmd_FailToStopUninhibit : BOOL;   // Program Command to Uninhibit Fail to Stop Alarm
   PCmd_IntlkTripAck : BOOL;   // Program Command to Acknowledge Interlock Trip Alarm
   PCmd_IntlkTripInhibit : BOOL;   // Program Command to Inhibit Interlock Trip Alarm
   PCmd_IntlkTripUninhibit : BOOL;   // Program Command to Uninhibit Interlock Trip Alarm
   PCmd_IOFaultAck : BOOL;   // Program Command to Acknowledge I/O Fault Alarm
   PCmd_IOFaultInhibit : BOOL;   // Program Command to Inhibit I/O Fault Alarm
   PCmd_IOFaultUninhibit : BOOL;   // Program Command to Uninhibit I/O Fault Alarm
   OCmd_Start : BOOL;   // Operator Command to Start Motor
   OCmd_Stop : BOOL;   // Operator Command to Stop Motor
   OCmd_Bypass : BOOL;   // Operator Command to Bypass all Bypassable Interlocks and Permissives
   OCmd_Check : BOOL;   // Operator Command to Check (not bypass) all Interlocks and Permissives
   MCmd_Disable : BOOL;   // Maintenance Command to Disable Motor
   MCmd_Enable : BOOL;   // Maintenance Command to Enable (allow to run) Motor
   OCmd_Reset : BOOL;   // Operator Command to Reset all Alarms requiring Reset
END_VAR
VAR_OUTPUT
   Out_Run : BOOL; {visible}   // 1=Run Motor, 0=Stop Motor
   Out_Start : BOOL; {visible}   // 1=Start Motor, 0=Motor left in current state
   Out_Stop : BOOL; {visible}   // 1=Stop Motor, 0=Motor left in current state
   Val_Owner : DINT;   // Current Object Owner ID (0=not owned)
   Val_Notify : SINT;   // Current Alarm Level and Acknowledgement (enumeration)
   Sts_Stopped : BOOL := 1; {visible}   // 1=Motor requested to stop and is confirmed stopped
   Sts_Starting : BOOL; {visible}   // 1=Motor requested to run and awaiting run feedback
   Sts_Running : BOOL; {visible}   // 1=Motor requested to run and is confirmed running
   Sts_Stopping : BOOL; {visible}   // 1=Motor requested to stop and awaiting stopped feedback
   Sts_Available : BOOL;   // 1=Motor available for control by automation (Prog)
   Sts_Bypass : BOOL;   // 1=Bypassable Interlocks and Permissives are Bypassed
   Sts_BypActive : BOOL;   // 1=Bypassing Active (Bypassed or Maintenance)
   Sts_Disabled : BOOL;   // 1=Motor is Disabled
   Sts_Err : BOOL; {visible}   // 1=Error in Config: see detail bits for reason
   Err_Timer : BOOL;   // 1=Error in Config: Start/Stop Check timer preset (use 0 to 2147483)
   Err_Sim : BOOL;   // 1=Error in Config: Simulation timer preset (use 0 to 2147483)
   Err_Alarm : BOOL;   // 1=Error in Config: Invalid Alarm Severity
   Sts_Hand : BOOL; {visible}   // 1=Mode is Hand (supersedes Maint, Ovrd, Prog, Oper)
   Sts_Maint : BOOL; {visible}   // 1=Mode is Maintenance (supersedes Ovrd, Prog, Oper)
   Sts_Ovrd : BOOL; {visible}   // 1=Mode is Override (supersedes Prog, Oper)
   Sts_Prog : BOOL; {visible}   // 1=Mode is Program (auto)
   Sts_Oper : BOOL := 1; {visible}   // 1=Mode is Operator (manual)
   Sts_ProgOperLock : BOOL;   // 1=Program or Operator has requested Mode Lock
   Sts_FailToStart : BOOL;   // 1=Motor Failed to Start (one-shot)
   Alm_FailToStart : BOOL;   // 1=Motor Fail to Start Alarm
   Ack_FailToStart : BOOL;   // 1=Fail to Start Alarm has been acknowledged
   Sts_FailToStartDisabled : BOOL;   // 1=Fail to Start Alarm has been disabled (will not be sent)
   Sts_FailToStartInhibited : BOOL;   // 1=Fail to Start Alarm has been inhibited by logic
   Sts_FailToStartSuppressed : BOOL;   // 1=Fail to Start Alarm has been suppressed (logged only)
   Sts_FailToStop : BOOL;   // 1=Motor Failed to Stop
   Alm_FailToStop : BOOL;   // 1=Motor Fail to Stop Alarm
   Ack_FailToStop : BOOL;   // 1=Fail to Stop Alarm has been acknowledged
   Sts_FailToStopDisabled : BOOL;   // 1=Fail to Stop Alarm has been disabled (will not be sent)
   Sts_FailToStopInhibited : BOOL;   // 1=Fail to Stop Alarm has been inhibited by logic
   Sts_FailToStopSuppressed : BOOL;   // 1=Fail to Stop Alarm has been suppressed (logged only)
   Sts_IntlkTrip : BOOL;   // 1=Motor stopped by an Interlock NOT OK (one-shot)
   Alm_IntlkTrip : BOOL;   // 1=Alarm: Motor stopped by an Interlock NOT OK
   Ack_IntlkTrip : BOOL;   // 1=Interlock Trip Alarm has been acknowledged
   Sts_IntlkTripDisabled : BOOL;   // 1=Interlock Trip Alarm is Disabled (not saved or sent)
   Sts_IntlkTripInhibited : BOOL;   // 1=Interlock Trip Alarm has been inhibited by logic
   Sts_IntlkTripSuppressed : BOOL;   // 1=Interlock Trip Alarm has been suppressed (logged only)
   Sts_IOFault : BOOL;   // I/O Comm Fault Status (0=OK, 1=Bad)
   Alm_IOFault : BOOL;   // 1=I/O Fault Alarm
   Ack_IOFault : BOOL;   // 1=I/O Fault Alarm has been acknowledged
   Sts_IOFaultDisabled : BOOL;   // 1=I/O Fault Alarm is Disabled (not saved or sent)
   Sts_IOFaultInhibited : BOOL;   // 1=I/O Fault Alarm has been inhibited by logic
   Sts_IOFaultSuppressed : BOOL;   // 1=I/O Fault Alarm has been suppressed (logged only)
   Rdy_Start : BOOL;   // 1=Ready to receive OCmd_Start (enables HMI button)
   Rdy_Stop : BOOL;   // 1=Ready to receive OCmd_Stop (enables HMI button)
   Rdy_Bypass : BOOL;   // 1=Ready to receive OCmd_Bypass (enables HMI button)
   Rdy_Check : BOOL;   // 1=Ready to receive OCmd_Check (enables HMI button)
   Rdy_Disable : BOOL;   // 1=Ready to receive MCmd_Disable (enables HMI button)
   Rdy_Enable : BOOL;   // 1=Ready to receive MCmd_Enable (enables HMI button)
   Rdy_Reset : BOOL;   // 1=Ready to receive OCmd_Reset (enables HMI button)
END_VAR
VAR
   Mode : P_Mode := (Cfg_PCmdClear := 1, Cfg_OvrdOverLock := 1, Sts_Oper := 1, Rdy_Rel := 1, Rdy_AcqLock := 1);   // Motor Mode Selection
   IOFault : P_Alarm := (Inp := 1, Cfg_AckReqd := 1, Cfg_Severity := 3, Ack := 1, Rdy_Disable := 1);   // I/O Fault Alarm
   IntlkTrip : P_Alarm := (Inp := 1, Cfg_AckReqd := 1, Cfg_Severity := 3, Ack := 1, Rdy_Disable := 1);   // Interlock Trip Alarm
   FailToStop : P_Alarm := (Inp := 1, Cfg_AckReqd := 1, Cfg_Severity := 3, Ack := 1, Rdy_Disable := 1);   // Motor Failed to Stop Alarm
   FailToStart : P_Alarm := (Inp := 1, Cfg_AckReqd := 1, Cfg_Severity := 3, Ack := 1, Rdy_Disable := 1);   // Motor Failed to Start Alarm
   Cfg_Tag : STRING_20 := 'P_Motor';   // Tagname for display on HMI
   Cfg_Label : STRING_20 := 'Motor Control';   // Label for graphic symbol displayed on HMI
   Cfg_Desc : STRING_40 := 'Single Speed Motor';   // Description for display on HMI
   Wrk_Run : BOOL;   // 1=Motor should be "running", 0=should be "stopped"
   Wrk_SimRunT : TIMER;   // Simulation Delay until Running
   Wrk_StopT : TIMER;   // Stop Check Timer
   Wrk_StartT : TIMER;   // Start Check Timer
   Wrk_Fault : BOOL;   // 1=a Motor Fault has been detected
   Wrk_SimStopT : TIMER;   // Simulation Delay until Stopped
   Wrk_RunFdbk : BOOL;   // Run Feedback based on mode, simulation, etc. 1=running
   Wrk_IntlkTrip : BOOL;   // 1=Interlock Not OK Tripped Running Motor
   Wrk_Notify : DINT;   // Buffer for building Val_Notify
   Wrk_Bypass : BOOL;   // Internal Bypassable Permissives and Interlocks are Bypassed flag
   Wrk_Disabled : BOOL;   // Internal Motor is Disabled
END_VAR

ROUTINE EnableInFalse   (* ladder *)
// Disabled is asserted; Outputs OFF; Run Status shown but Alarms disabled
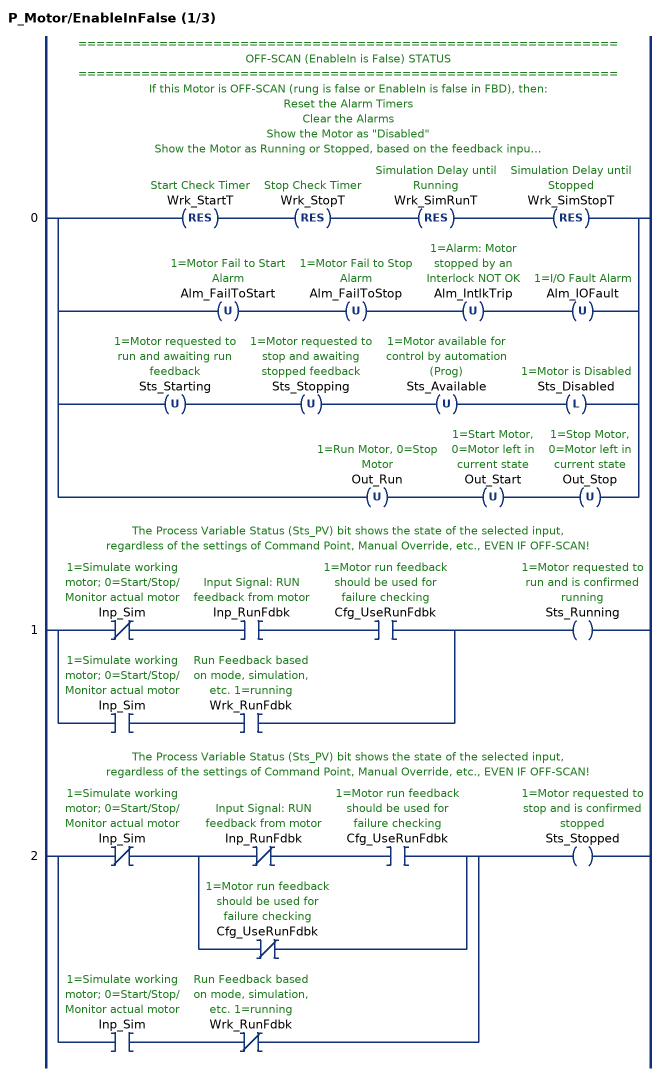
   // ============================================================
   // OFF-SCAN (EnableIn is False) STATUS
   // ============================================================
   // If this Motor is OFF-SCAN (rung is false or EnableIn is false in FBD), then:
   // Reset the Alarm Timers
   // Clear the Alarms
   // Show the Motor as "Disabled"
   // Show the Motor as Running or Stopped, based on the feedback input
   // Turn off the Outputs
   // Other data are left in Last State!
   0: [RES(Wrk_StartT) RES(Wrk_StopT) RES(Wrk_SimRunT) RES(Wrk_SimStopT) ,OTU(Alm_FailToStart) OTU(Alm_FailToStop) OTU(Alm_IntlkTrip) OTU(Alm_IOFault) ,OTU(Sts_Starting) OTU(Sts_Stopping) OTU(Sts_Available) OTL(Sts_Disabled) ,OTU(Out_Run) OTU(Out_Start) OTU(Out_Stop) ];
   // The Process Variable Status (Sts_PV) bit shows the state of the selected input,
   // regardless of the settings of Command Point, Manual Override, etc., EVEN IF OFF-SCAN!
   1: [XIO(Inp_Sim) XIC(Inp_RunFdbk) XIC(Cfg_UseRunFdbk) ,XIC(Inp_Sim) XIC(Wrk_RunFdbk) ]OTE(Sts_Running);
   // The Process Variable Status (Sts_PV) bit shows the state of the selected input,
   // regardless of the settings of Command Point, Manual Override, etc., EVEN IF OFF-SCAN!
   2: [XIO(Inp_Sim) [XIO(Inp_RunFdbk) XIC(Cfg_UseRunFdbk) ,XIO(Cfg_UseRunFdbk) ] ,XIC(Inp_Sim) XIO(Wrk_RunFdbk) ]OTE(Sts_Stopped);
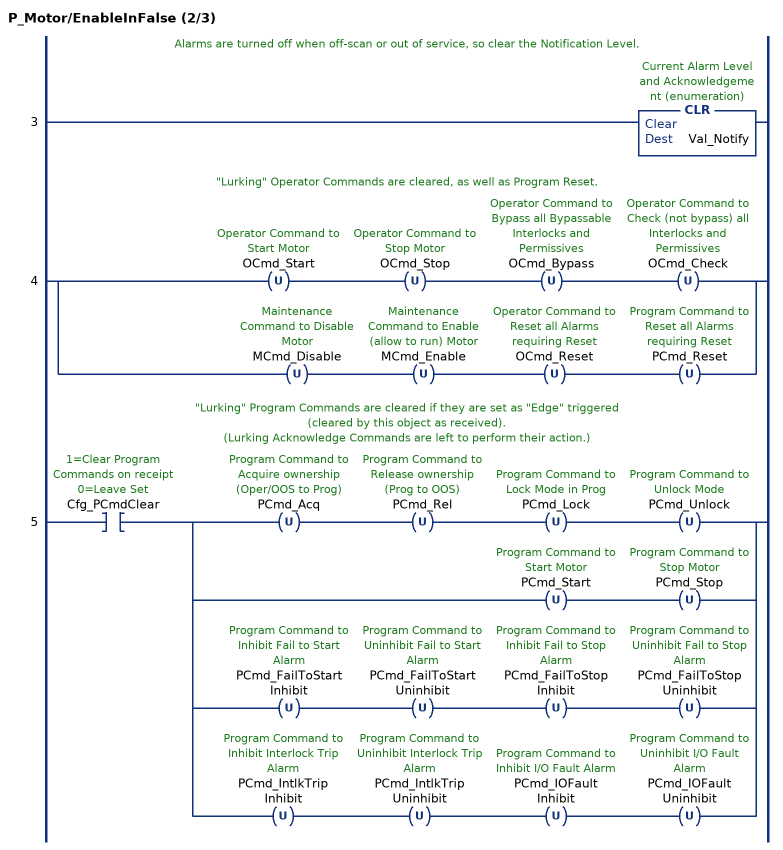
   // Alarms are turned off when off-scan or out of service, so clear the Notification Level.
   3: CLR(Val_Notify);
   // "Lurking" Operator Commands are cleared, as well as Program Reset.
   4: [OTU(OCmd_Start) OTU(OCmd_Stop) OTU(OCmd_Bypass) OTU(OCmd_Check) ,OTU(MCmd_Disable) OTU(MCmd_Enable) OTU(OCmd_Reset) OTU(PCmd_Reset) ];
   // "Lurking" Program Commands are cleared if they are set as "Edge" triggered
   // (cleared by this object as received).
   // (Lurking Acknowledge Commands are left to perform their action.)
   5: XIC(Cfg_PCmdClear)[OTU(PCmd_Acq) OTU(PCmd_Rel) OTU(PCmd_Lock) OTU(PCmd_Unlock) ,OTU(PCmd_Start) OTU(PCmd_Stop) ,OTU(PCmd_FailToStartInhibit) OTU(PCmd_FailToStartUninhibit) OTU(PCmd_FailToStopInhibit) OTU(PCmd_FailToStopUninhibit) ,OTU(PCmd_IntlkTripInhibit) OTU(PCmd_IntlkTripUninhibit) OTU(PCmd_IOFaultInhibit) OTU(PCmd_IOFaultUninhibit) ];
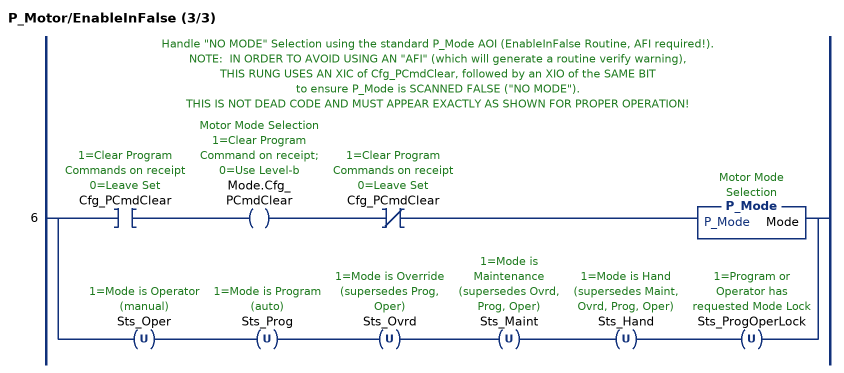
   // Handle "NO MODE" Selection using the standard P_Mode AOI (EnableInFalse Routine, AFI required!).
   // NOTE:  IN ORDER TO AVOID USING AN "AFI" (which will generate a routine verify warning),
   // THIS RUNG USES AN XIC of Cfg_PCmdClear, followed by an XIO of the SAME BIT
   // to ensure P_Mode is SCANNED FALSE ("NO MODE").
   // THIS IS NOT DEAD CODE AND MUST APPEAR EXACTLY AS SHOWN FOR PROPER OPERATION!
   6: [XIC(Cfg_PCmdClear) OTE(Mode.Cfg_PCmdClear) XIO(Cfg_PCmdClear) P_Mode(Mode) ,OTU(Sts_Oper) OTU(Sts_Prog) OTU(Sts_Ovrd) OTU(Sts_Maint) OTU(Sts_Hand) OTU(Sts_ProgOperLock) ];
END_ROUTINE
